(* IEC 61131-3 sources: xPLCCore/codesys_code/Application/Robot_FBs/AxisGroupManager_BB, 5 files *)

(* ---- AxisGroupManager_BB.st ---- *)
//==============================================================================
// Main Function Block Definition
//==============================================================================
FUNCTION_BLOCK AxisGroupManager_BB

VAR
    // --- Internal State & Events ---
    _preState : E_RobotState := E_RobotState.NULL;
    _eState : E_RobotState := E_RobotState.NULL;
    _nxtState : E_RobotState := E_RobotState.NULL;

    _eCurrentEvent : E_RobotEvent := E_RobotEvent.EV_NONE; // Holds the event to be processed

    // --- Axis Configuration ---
    _agAxisGroup : REFERENCE TO AXIS_GROUP_REF_SM3; // Internal reference to the axis group

    // --- Status & Error Info ---
    _bIsHomed : BOOL;
    _bIsInError : BOOL;
    _dwErrorID : DWORD;
    _bReadyForOperation : BOOL;

    // --- Motion Control Function Blocks ---
    _fbPower : MC_Power;
    _fbGroupEnable : MC_GroupEnable;
    _fbGroupReset : MC_GroupReset;
    _fbGroupDisable : MC_GroupDisable;
    _fbHome : MC_Home;

	SMC_GroupPower_0:SM3_Robotics.SMC_GroupPower;
	GroupPower_Flag:BOOL:=FALSE;
	//SMC_GroupReset_0:SM3_Robotics.MC_GroupReset;
	SMC_GroupDisable:SM3_Robotics.MC_GroupDisable;

	SMC_GroupReset:SM3_Robotics.MC_GroupReset;

	enable_fb:SM3_Robotics.MC_GroupEnable;

	homing_fb:FB_Homing;

	MoveLinearAbsolute_0: SM3_Robotics.MC_MoveLinearAbsolute;
	motionPoseRunPass:INT;
	motionPoseIdx:INT;

	stateCD:INT;

END_VAR
(* =========== IMPLEMENTATION =========== *)

(* ---- FB_init.st ---- *)
//==============================================================================
// FB_init: Called once on startup to configure the FB instance.
//==============================================================================
METHOD FB_init : BOOL
VAR_INPUT
    bInitRetains : BOOL; // This parameter is required by the compiler
    bInCopyCode : BOOL;  // This parameter is required by the compiler

    // The robot's axis group
    agAxisGroup : REFERENCE TO AXIS_GROUP_REF_SM3;

END_VAR
VAR
    i : UINT;
END_VAR
(* =========== IMPLEMENTATION =========== *)

// Store the reference to the axis group
_agAxisGroup REF= agAxisGroup;

FB_init := TRUE;

_eState:=E_RobotState.NULL;
_nxtState:=E_RobotState.UnInited;
Update(1);//exit old state
_preState:=_eState;
_eState:=_nxtState;
Update(-1);//enter new state

(* ---- Transition.st ---- *)
METHOD Transition : BOOL
VAR_INPUT
    eEvent : E_RobotEvent;
END_VAR
VAR_OUTPUT
	error:BOOL;
	new_state:E_RobotState;
END_VAR
(* =========== IMPLEMENTATION =========== *)

new_state:=_eState;
CASE _eState OF
	E_RobotState.UnInited:
		CASE eEvent OF
			E_RobotEvent.EV_POWER_ON:
			 new_state:=E_RobotState.Powering;
		END_CASE

	E_RobotState.Powering:
		CASE eEvent OF
			E_RobotEvent.EV_POWER_OFF,
			E_RobotEvent.EV_ERROR,
			E_RobotEvent.EV_RESET:
			   new_state:=E_RobotState.UnInited;
			E_RobotEvent.EV_OK:
			   new_state:=E_RobotState.Powered;
		END_CASE
	E_RobotState.Powered:
		CASE eEvent OF
		E_RobotEvent.EV_GROUP_ENABLE:
			 new_state:=E_RobotState.GroupEnabling;
		END_CASE

	E_RobotState.GroupEnabling:
		CASE eEvent OF
		E_RobotEvent.EV_OK:
			 new_state:=E_RobotState.GroupEnabled;
		END_CASE

	E_RobotState.GroupEnabled:
		CASE eEvent OF
		E_RobotEvent.EV_HOME_GO:
			 new_state:=E_RobotState.Homing;
		E_RobotEvent.EV_HOME_GO_FORCE_SKIP:
			 new_state:=E_RobotState.Ready;
		END_CASE
	E_RobotState.Homing:
		CASE eEvent OF
		E_RobotEvent.EV_OK:
			 new_state:=E_RobotState.Ready;
		END_CASE

	E_RobotState.Ready:
		CASE eEvent OF
		E_RobotEvent.EV_HOME_GO:
			 new_state:=E_RobotState.Homing;
		END_CASE

	E_RobotState.Error:
		CASE eEvent OF
		E_RobotEvent.EV_RESET:
			 new_state:=E_RobotState.UnInited;
		END_CASE

END_CASE

IF(new_state=_eState)THEN//error/stop handling
	IF(eEvent=E_RobotEvent.EV_ERROR)THEN
		new_state:=E_RobotState.Error;
	END_IF

END_IF

IF(new_state<>_eState)THEN
  _nxtState:=new_state;
  Update(1);//exit old state
  _preState:=_eState;
  _eState:=_nxtState;
  Update(-1);//enter new state

END_IF

(* ---- Update.st ---- *)
METHOD Update : BOOL
VAR_INPUT
	//-1 enter, 0 update,1 exit current(_eState) state
	uidx:INT:=0;
END_VAR
VAR

END_VAR
(* =========== IMPLEMENTATION =========== *)
Update:=TRUE;

CASE _eState OF
	E_RobotState.UnInited:
		IF(uidx=-1)THEN//enter
			GroupPower_Flag:=FALSE;
			SMC_GroupDisable(
				AxisGroup:=_agAxisGroup,
				Execute:=FALSE
			);

			SMC_GroupReset(
				AxisGroup:=_agAxisGroup,
				Execute:=FALSE
				);

			IoConfig_Globals.EtherCAT_Master_SoftMotion.xRestart:=TRUE;

			IoConfig_Globals.EtherCAT_Master_SoftMotion();
			(*MotorReset(
			Axis:=IoConfig_Globals.EAxis1,
			Execute:=FALSE);*)

		END_IF
		IF(uidx=0)THEN//update
			SMC_GroupDisable(
				AxisGroup:=_agAxisGroup,
				Execute:=TRUE
			);
			SMC_GroupReset(
				AxisGroup:=_agAxisGroup,
				Execute:=TRUE
				);
			IoConfig_Globals.EtherCAT_Master_SoftMotion();

			IoConfig_Globals.EtherCAT_Master_SoftMotion.xRestart:=FALSE;

			(*MotorReset(
			Axis:=IoConfig_Globals.EAxis1,
			Execute:=TRUE);*)

		END_IF
		RETURN;
	E_RobotState.Powering:
		IF(uidx=-1)THEN//enter
			GroupPower_Flag:=FALSE;
		ELSIF(uidx=0)THEN
			GroupPower_Flag:=TRUE;
			IF(SMC_GroupPower_0.Status) THEN
				Transition(E_RobotEvent.EV_OK);
			END_IF
		//ELSIF(uidx=1)THEN

		END_IF
	//E_RobotState.Powered://a halt state, wait for user
		//RETURN;
	E_RobotState.GroupEnabling:

		IF(uidx=-1)THEN//enter
			enable_fb(
			AxisGroup:=_agAxisGroup,
			Execute:=FALSE,
			);
		ELSIF(uidx=0)THEN
			enable_fb(
			AxisGroup:=_agAxisGroup,
			Execute:=TRUE,
			);

			IF(enable_fb.Done) THEN
				Transition(E_RobotEvent.EV_OK);
			END_IF
		END_IF

	//E_RobotState.GroupEnabled://a halt state, wait for user's next event
		//RETURN;

	E_RobotState.Homing:

		IF(uidx=-1)THEN//enter
			homing_fb(
			bExecute:=FALSE,
			);
			stateCD:=100;
		ELSIF(uidx=0)THEN

			homing_fb(
			bExecute:=TRUE,
			);
			IF(homing_fb.bDone) THEN

				stateCD:=stateCD-1;
				IF(stateCD=0)THEN
					Transition(E_RobotEvent.EV_OK);
				END_IF
			ELSE

				stateCD:=100;
			END_IF

		ELSIF(uidx=1)THEN

			homing_fb(
			bExecute:=FALSE,
			);

		END_IF

	E_RobotState.Ready:

		IF(uidx=-1)THEN//enter
		ELSIF(uidx=0)THEN
			uidx:=uidx;

		END_IF

	E_RobotState.Error:

		IF(uidx=-1)THEN//enter
			GroupPower_Flag:=FALSE;
			SMC_GroupDisable(
				AxisGroup:=_agAxisGroup,
				Execute:=FALSE
			);

			SMC_GroupReset(
				AxisGroup:=_agAxisGroup,
				Execute:=FALSE
				);

			(*MotorReset(
			Axis:=IoConfig_Globals.EAxis1,
			Execute:=FALSE);*)

		END_IF
		IF(uidx=0)THEN//enter
			SMC_GroupDisable(
				AxisGroup:=_agAxisGroup,
				Execute:=TRUE
			);
			SMC_GroupReset(
				AxisGroup:=_agAxisGroup,
				Execute:=TRUE
				);

			(*MotorReset(
			Axis:=IoConfig_Globals.EAxis1,
			Execute:=TRUE);*)

		END_IF

END_CASE

SMC_GroupPower_0(
AxisGroup:=_agAxisGroup,
Enable:=TRUE,
bRegulatorOn:=GroupPower_Flag,
bDriveStart:=GroupPower_Flag
);

(* ---- Update_1.st ---- *)
METHOD Update_1 : BOOL
VAR_INPUT
	//-1 enter, 0 update,1 exit current(_eState) state
	uidx:INT:=0;
END_VAR
VAR

RunSpeed:REAL:=100000;
RunFactor:REAL:=1;

	motionPoses:ARRAY[0..3] OF  SM3_Robotics.SMC_POS_REF :=
    [ ( c := (x := 60.0, y := -60.0, z := -10.0, a := 0.0)),
	 ( c := (x := 60.0, y := 60.0, z := -10.0, a := 0.0)),
	  ( c := (x := -60.0, y := 60.0, z := -10.0, a := 0.0)),
	   ( c := (x := -60.0, y := -60.0, z := -10.0, a := 0.0))

	];
	TransitionParameter:ARRAY [0..1]OF LREAL:=[2,0];
END_VAR
(* =========== IMPLEMENTATION =========== *)
Update_1:=TRUE;

CASE _eState OF
	E_RobotState.UnInited:
	    IF(uidx=1)THEN
			//EXIT, you may do some init stuff here
		END_IF
		RETURN;
	E_RobotState.Powering:
		IF(uidx=-1)THEN//enter
			GroupPower_Flag:=FALSE;
		ELSIF(uidx=0)THEN
			GroupPower_Flag:=TRUE;
			IF(SMC_GroupPower_0.Status) THEN
				Transition(E_RobotEvent.EV_OK);
			END_IF
		//ELSIF(uidx=1)THEN

		END_IF
	//E_RobotState.Powered://a halt state, wait for user
		//RETURN;
	E_RobotState.GroupEnabling:

		IF(uidx=-1)THEN//enter
			enable_fb(
			AxisGroup:=_agAxisGroup,
			Execute:=FALSE,
			);
		ELSIF(uidx=0)THEN
			enable_fb(
			AxisGroup:=_agAxisGroup,
			Execute:=TRUE,
			);

			IF(enable_fb.Done) THEN
				Transition(E_RobotEvent.EV_OK);
			END_IF
		END_IF

	//E_RobotState.GroupEnabled://a halt state, wait for user's next event
		//RETURN;

	E_RobotState.Homing:

		IF(uidx=-1)THEN//enter
			homing_fb(
			bExecute:=FALSE,
			);
			stateCD:=100;
		ELSIF(uidx=0)THEN

			homing_fb(
			bExecute:=TRUE,
			);
			IF(homing_fb.bDone) THEN

				stateCD:=stateCD-1;
				IF(stateCD=0)THEN
					Transition(E_RobotEvent.EV_OK);
				END_IF
			ELSE

				stateCD:=100;
			END_IF

		ELSIF(uidx=1)THEN

			homing_fb(
			bExecute:=FALSE,
			);

		END_IF

	E_RobotState.Ready:

		IF(uidx=-1)THEN//enter
			motionPoseIdx:=0;
			motionPoseRunPass:=0;
		ELSIF(uidx=0)THEN

			MoveLinearAbsolute_0(
			AxisGroup          := _agAxisGroup,
			Execute            := 0
			);

			IF(motionPoseIdx>3)THEN
				IF(motionPoseRunPass<1)THEN
					motionPoseRunPass:=motionPoseRunPass+1;
					motionPoseIdx:=0;
				END_IF
			ELSE

				MoveLinearAbsolute_0(
				AxisGroup          := _agAxisGroup,
				Execute            := 1,
				Position           := motionPoses[motionPoseIdx],              // ← [0.0,0.0,0.0,0.0]
				Velocity           := RunSpeed,                 // 速度 (mm/s 或 deg/s)
				Acceleration       := RunSpeed,                // 加速度 (mm/s² 或 deg/s²)
				Deceleration       := RunSpeed,
				Jerk               := RunSpeed*5,
				CoordSystem		   := SMC_COORD_SYSTEM.MCS,

				BufferMode         := SM3_Common.MC_BUFFER_MODE.BlendingHigh, // 緩衝模式
				TransitionMode     := SM3_Robotics.MC_TRANSITION_MODE.TMCornerDistance,
				TransitionParameter:= TransitionParameter,

				//BufferMode         := SM3_Common.MC_BUFFER_MODE.Buffered,
				//TransitionMode     := SM3_Robotics.MC_TRANSITION_MODE.TMNone,

				VelFactor:=RunFactor,
				AccFactor:=RunFactor,
				JerkFactor:=RunFactor,
				TorqueFactor:=1,
				Done=>,
				Busy=>,
				Active=>,
				Error=>,
				ErrorID=>,
				MovementId=>
				);

				motionPoseIdx:=motionPoseIdx+1;

			END_IF

		END_IF

	E_RobotState.Error:

		IF(uidx=-1)THEN//enter
			GroupPower_Flag:=FALSE;
			SMC_GroupDisable(
				AxisGroup:=_agAxisGroup,
				Execute:=FALSE
			);

			SMC_GroupReset(
				AxisGroup:=_agAxisGroup,
				Execute:=FALSE
				);
		END_IF
		IF(uidx=0)THEN//enter
			SMC_GroupDisable(
				AxisGroup:=_agAxisGroup,
				Execute:=TRUE
			);
			SMC_GroupReset(
				AxisGroup:=_agAxisGroup,
				Execute:=TRUE
				);

		END_IF

END_CASE

SMC_GroupPower_0(
AxisGroup:=_agAxisGroup,
Enable:=TRUE,
bRegulatorOn:=GroupPower_Flag,
bDriveStart:=GroupPower_Flag
);
